FUNCTION_BLOCK FB_MachineControl EXTENDS FB_BaseTopElement IMPLEMENTS ITF_MachineControlConfigure
VAR
	(*	Inicjalizacja		*)
	bInitializeCycle			: BOOL;
	bInitDone					: BOOL;
	(*	Konfiguracja		*)
	itfMachineConfigure			: ITF_MachineConfigure;		//moduł konfiguracji
	(*	TopElementu systemu	*)
	arrTopElements					: ARRAY [0..GVL_BaseConstans.MAX_NUMBER_OF_TOP_ELEMENT] OF ITF_BaseTopElement;
	iNumberOfAddedTopElement		: INT := -1;//przy dodawaniu element 0 to system 
	uiNumberOfAllAddedElements		: UINT;		//liczba elementow które są na maszynie 
	(*	Master komunikatora dla top elementów maszyny	*)
	fbMasterCommunicator			: FB_BaseCommunicator;
	(*	Zarządzenia stanami i trybami pracy	*)
	itfSaMController				: ITF_SaMController;
	(*	Stany i Tryby	*)
	arrRequestChangeState			: ARRAY [1..GVL_SaMConstans.NUMBER_OF_COMMAND_CHANGE_STATES] OF ITF_IOButton;	
	arrRequestChangeMode			: ARRAY [1..GVL_SaMConstans.NUMBER_OF_COMMAND_CHANGE_MODES] OF ITF_IOButton;
END_VAR

IF (NOT THIS^.bInitializeCycle) THEN
	THIS^.bInitializeCycle		:= TRUE;
	THIS^.bInitDone				:= THIS^.InitializeCycle ();
ELSIF (THIS^.bInitDone) THEN
	THIS^.ExecuteCycle ();
END_IF

(*			
	EVERDE sp. z o.o.
	Rafał Osajda		29.10.2025		TC 4024.66
	Dodawanie intefejsu konfiguracji
*)
METHOD PUBLIC AddModulConfigure : BOOL
VAR_INPUT
	fbMachineConfigure			: ITF_MachineConfigure;
END_VAR
THIS^.itfMachineConfigure		:= fbMachineConfigure;
END_METHOD

METHOD PUBLIC AddModulSaM : BOOL
VAR_INPUT
	fbSaMController			: ITF_SaMController;
END_VAR
THIS^.itfSaMController		:= fbSaMController;
THIS^.AddControlElement (itfControlElement	:= fbSaMController);
END_METHOD

METHOD PUBLIC AddRequestModeChange : BOOL
VAR_INPUT
	iNumberOfRequest			: INT;
	itfRequest					: ITF_IOButton;
END_VAR
THIS^.arrRequestChangeMode [iNumberOfRequest]	:= itfRequest;
END_METHOD

METHOD PUBLIC AddRequestStateChange : BOOL
VAR_INPUT
	iNumberOfRequest			: INT;
	itfRequest					: ITF_IOButton;
END_VAR
THIS^.arrRequestChangeState [iNumberOfRequest]	:= itfRequest;
END_METHOD

(*			
	EVERDE sp. z o.o.
	Rafał Osajda		29.10.2025		TC 4024.66
	Metoda dodawania top elementu wywoływana z konfiguracji
*)
METHOD AddTopElementFromConfiguration : BOOL
VAR_INPUT
	fbTopElement		: ITF_BaseTopElement;
END_VAR
IF (THIS^.iNumberOfAddedTopElement + 1 <= TO_INT (GVL_BaseConstans.MAX_NUMBER_OF_TOP_ELEMENT)) THEN
	THIS^.iNumberOfAddedTopElement							:= THIS^.iNumberOfAddedTopElement + 1;
	THIS^.arrTopElements [THIS^.iNumberOfAddedTopElement]	:= fbTopElement;
	
	THIS^.arrTopElements [THIS^.iNumberOfAddedTopElement].LinkCommonData (stCommonData	:= THIS^.refstCommonData);
	THIS^.arrTopElements [THIS^.iNumberOfAddedTopElement].LinkSS1 (fbSS1	:= THIS^.itfSS1);
	THIS^.arrTopElements [THIS^.iNumberOfAddedTopElement].LinkSTO (fbSTO	:= THIS^.itfSTO);
	THIS^.arrTopElements [THIS^.iNumberOfAddedTopElement].LinkCommunicator (fbCommunicator	:= THIS^.fbMasterCommunicator);
	(*	Podpięcie systemu sterowania stanami i trybami	*)
//	THIS^.arrTopElements [THIS^.iNumberOfAddedTopElement].LinkSAM (fbSAM	:= THIS^. tu będzie interfijs do SITP);
	THIS^.arrTopElements [THIS^.iNumberOfAddedTopElement].FirstCycle ();
	THIS^.uiNumberOfAllAddedElements 						:= THIS^.arrTopElements [THIS^.iNumberOfAddedTopElement].SetID (uiID := THIS^.uiNumberOfAllAddedElements + 1);
	THIS^.refstCommonData.itfLogger.SetNumerOfReportsIntheSystem (
			uiValue := THIS^.arrTopElements [THIS^.iNumberOfAddedTopElement].SetEventsIDs (
				uiNewID := THIS^.refstCommonData.itfLogger.GetNumerOfReportsIntheSystem ()
			)
	);
	THIS^.arrTopElements [THIS^.iNumberOfAddedTopElement].SetCode (sCode := '0.0.0.0.0', sAdd := TO_STRING (THIS^.iNumberOfAddedTopElement));
	
	AddTopElementFromConfiguration							:= TRUE;
END_IF
END_METHOD

METHOD PRIVATE ExecuteCycle

VAR
	iI: INT;
END_VAR
	(*	Zarządzanie Stanami i Trybami	*)

THIS^.ExecuteCycle_SaM ();

	(*	Wywołanie metod obsługiwanych co cykl dla każdego elementu	*)

FOR iI := 0 TO THIS^.iNumberOfAddedTopElement DO
	THIS^.arrTopElements [iI].ExecuteEveryCycle_Test ();
	THIS^.arrTopElements [iI].ExecuteEveryCycle_Operation ();
	THIS^.arrTopElements [iI].ExecuteEveryCycle_Status ();
	THIS^.arrTopElements [iI].ExecuteEveryCycle_Error ();
	
END_FOR
END_METHOD

METHOD PRIVATE ExecuteCycle_SaM
VAR
	iI					: INT;
END_VAR

	(*	Zarządzanie stanami i trybami pracy 	*)

	(*	Testowanie czy jest rządzanie zmiany trybu	*)
FOR iI := 1 TO 10 DO 
	IF (THIS^.arrRequestChangeMode [iI] <> 0) THEN
		IF (THIS^.arrRequestChangeMode [iI].IsPressed ()) THEN
			THIS^.itfSaMController.Execute (iNumberOfCommand := iI, eChangeCategory := E_SaMChangeCategory.eMode);
		END_IF
	END_IF
END_FOR	
	
	(*	Testowanie czy jest rządanie zmiany stany	*)
FOR iI := 1 TO 10 DO 
	IF (THIS^.arrRequestChangeState [iI] <> 0) THEN
		IF (THIS^.arrRequestChangeState [iI].IsPressed ()) THEN
			THIS^.itfSaMController.Execute (iNumberOfCommand := iI, eChangeCategory := E_SaMChangeCategory.eState);
		END_IF
	END_IF
END_FOR
	

IF (NOT THIS^.itfSaMController.IsChangeModeBusy () AND NOT THIS^.itfSaMController.IsChangeStateBusy ()) THEN
	;
END_IF

	(*	Obsługa stanów aktywnych - ing	*)
	
	(*	Obsługa stanów biernych		*)
END_METHOD

METHOD PRIVATE InitializeCycle : BOOL
VAR
	bResult					: BOOL;
	iI: INT;
END_VAR
bResult				:= TRUE;

bResult				:= bResult AND THIS^.itfMachineConfigure.Configure (fbMachineControl := THIS^);

//FOR iI := 0 TO THIS^.iNumberOfAddedTopElement DO
//	bResult				:= bResult AND THIS^.arrTopElements [iI].FirstCycle ();
//END_FOR



InitializeCycle		:= bResult;
END_METHOD

END_FUNCTION_BLOCK

(* stored: Version 1.1.0.1
   POU FB_MachineControl: Id {03d9ff00-a300-4d9d-a349-75e3318a4c90}, SpecialFunc None
   Folder ITF_MachineControlConfigure: Id {973d3ff0-85f0-4bae-9395-cc62a4917833}
   Folder WiazanieModulow: Id {3d8e3574-09c0-0f20-0429-cf1b0f8aec79}
   Method AddModulConfigure: Id {e05e86ab-e65a-0460-123e-9f866e36dccc}
   Method AddModulSaM: Id {fdfb6f32-ad29-05b9-1f5f-f81a0f2962ac}
   Method AddRequestModeChange: Id {eee38abc-f39d-0ce2-0412-12f1dcddd8de}
   Method AddRequestStateChange: Id {3a316008-6053-0642-3d72-eda4def5bdc4}
   Method AddTopElementFromConfiguration: Id {100f011a-3941-0f6f-14c0-c4dea046c178}
   Method ExecuteCycle: Id {7066db40-c8ea-4d9b-9b50-7a0d826fe39e}
   Method ExecuteCycle_SaM: Id {111ca252-3465-079b-3f8c-a42b1dc9a298}
   Method InitializeCycle: Id {f127c58d-f380-4c5b-91fc-37aed1ddc70f} *)
